{attribute 'analysis' := '-33'}
PROGRAM INTERNAL PRG_WritingPrimitiveTests
{IF defined (UNIT_TEST)}
    fbEncodeZigZag32Tests       : FB_EncodeZigZag32Tests;
    fbEncodeZigZag64Tests       : FB_EncodeZigZag64Tests;
    fbWriteStringTests          : FB_WriteStringTests;
    fbWriteTagTests             : FB_WriteTagTests;
    fbWriteBytesTests           : FB_WriteBytesTests;
    fbWriteFloatTests           : FB_WriteFloatTests;
    fbWriteDoubleTests           : FB_WriteDoubleTests;
{END_IF}

END_PROGRAM

(* stored: Version 1.1.0.1
   POU PRG_WritingPrimitiveTests: Id {50edbeac-899e-4307-aeca-b3f79972fc27}, SpecialFunc None *)
